PROGRAM CraneSteering
VAR
	fbMotionRefGen : FB_MotionReferenceGenerator;
	
END_VAR

END_PROGRAM

(* stored: Version 1.1.0.1, ProductVersion 3.1.4024.10
   POU CraneSteering: Id {11a0f5e4-dc13-4aac-aeaa-4d3c9914c435}, SpecialFunc None *)
